// TwinCAT 3 PLC project Untitled1
// ProgramVersion: 3.1.4023.0
// libraries:
//   Tc2_Standard, * (Beckhoff Automation GmbH)
//   Tc2_System, * (Beckhoff Automation GmbH)
//   Tc3_EventLogger, * (Beckhoff Automation GmbH)
//   Tc3_Module, * (Beckhoff Automation GmbH)
//   VisuDialogs, * (System)
//   VisuSymbols,3.5.10.0,System
// project tree:
//   / GlobalTextList.TcGTLO (not stored), PlcTask.TcTTO (not stored), Visualization Manager.TcVMO (not stored)
//   POUs/ MAIN.TcPOU
// real-time tasks:
//   TASK PlcTask: cycle T#10ms, priority 20, ADS port 350
// I/O:
//   DEVICE Device 1 (EtherCAT), AmsNetId 5.112.67.239.2.1
//     Term 7 (EK1200) [EK1200-5000 EtherCAT Power supply (2A E-Bus)]
//       Term 2 (EL4004) [EL4004 4Ch. Ana. Output 0-10V, 12bit]
//       Term 3 (EL4004) [EL4004 4Ch. Ana. Output 0-10V, 12bit]
//       Term 8 (EL3024) [EL3024 4Ch. Ana. Input 4-20mA DIFF]
//       Term 9 (EL3024) [EL3024 4Ch. Ana. Input 4-20mA DIFF]
//       Term 12 (EL1859) [EL1859 8Ch. Dig. Input 24V, 3ms, 8Ch. Dig. Output 24V, 0.5A]
//       Term 13 (EL9011) [EL9011 End Terminal]
// variable links:
//   Untitled1/Untitled1 Instance <-> Device 1 (EtherCAT)/Term 7 (EK1200)/Term 12 (EL1859)
//     PlcTask Inputs/MAIN.EMERGENCY_STOP <-> Channel 1/EMERGENCY STOP
//     PlcTask Inputs/MAIN.Start_Button <-> Channel 2/Start Button
//     PlcTask Inputs/MAIN.Stop_Button <-> Channel 3/Stop Button
//     PlcTask Outputs/MAIN.Motor_Direction <-> Channel 10/Motor Direction
//     PlcTask Outputs/MAIN.Motor_ON_OFF <-> Channel 9/Motor ON/OFF
//   Untitled1/Untitled1 Instance <-> Device 1 (EtherCAT)/Term 7 (EK1200)/Term 2 (EL4004)
//     PlcTask Outputs/MAIN.Flow_Valve_1 <-> AO Outputs Channel 4/Flow_Valve_1
//     PlcTask Outputs/MAIN.Level_Valve_1 <-> AO Outputs Channel 1/Level_Valve_1
//     PlcTask Outputs/MAIN.Level_Valve_2 <-> AO Outputs Channel 2/Level_Valve_2
//     PlcTask Outputs/MAIN.Level_Valve_3 <-> AO Outputs Channel 3/Level_Valve_3
//   Untitled1/Untitled1 Instance <-> Device 1 (EtherCAT)/Term 7 (EK1200)/Term 3 (EL4004)
//     PlcTask Outputs/MAIN.Gas_Valve <-> AO Outputs Channel 1/Gas_Valve
//     PlcTask Outputs/MAIN.Mixer_Valve <-> AO Outputs Channel 2/Mixer_Valve
//     PlcTask Outputs/MAIN.Motor_speed <-> AO Outputs Channel 3/Motor_Speed
//   Untitled1/Untitled1 Instance <-> Device 1 (EtherCAT)/Term 7 (EK1200)/Term 8 (EL3024)
//     PlcTask Inputs/MAIN.Pressure_Differencial_Transmitter_1 <-> AI Standard Channel 1/PDT 1
//     PlcTask Inputs/MAIN.Pressure_Differencial_Transmitter_2 <-> AI Standard Channel 3/PDT 2
//     PlcTask Inputs/MAIN.Pressure_Transmitter_1 <-> AI Standard Channel 2/PT 1
//     PlcTask Inputs/MAIN.Pressure_Transmitter_3 <-> AI Standard Channel 4/PT 3
//   Untitled1/Untitled1 Instance <-> Device 1 (EtherCAT)/Term 7 (EK1200)/Term 9 (EL3024)
//     PlcTask Inputs/MAIN.Level_Transmitter_1 <-> AI Standard Channel 2/ Level Transmitter 1
//     PlcTask Inputs/MAIN.Level_Transmitter_2 <-> AI Standard Channel 3/Level Transmitter 2
//     PlcTask Inputs/MAIN.Pressure_Transmitter_2 <-> AI Standard Channel 1/PT 2
//     PlcTask Inputs/MAIN.Temperature_Transmitter <-> AI Standard Channel 4/Temperature Transmitter

// ---- POUs/MAIN.TcPOU
PROGRAM MAIN
VAR
	//Linking variables to IO cards
	Flow_Valve_1 AT %Q* : INT;
	Level_Valve_1 AT %Q* : INT;
	Level_Valve_2 AT %Q* : INT;
	Level_Valve_3 AT %Q* : INT;
	Gas_Valve AT %Q* : INT;
	Mixer_Valve AT %Q* : INT;
	Motor_speed AT %Q* : INT;
	Motor_ON_OFF AT %Q* :BOOL;
	Motor_Direction AT %Q* :BOOL; 
	Start_Button AT %I* :BOOL;
	Stop_Button AT %I* : BOOL; 
	EMERGENCY_STOP AT %I* : BOOL; 
	Level_Transmitter_1 AT %I* :INT; 
	Level_Transmitter_2 AT %I* :INT; 
	Temperature_Transmitter AT %I* :INT;  
	Pressure_Differencial_Transmitter_1 AT %I* : INT;
	Pressure_Differencial_Transmitter_2 AT %I* : INT;
	Pressure_Transmitter_1 AT %I* : INT ; 
	Pressure_Transmitter_2 AT %I* : INT ; 
	Pressure_Transmitter_3 AT %I* : INT ; 

	
	//User Input as percentage
	Flow_Valve_1_Percentage: INT :=100;
	Level_Valve_1_Percentage: INT    ;
	Level_Valve_2_Percentage: INT;
	Level_Valve_3_Percentage: INT;
	Motor_speed_Percentage: INT; 
	Motor_ON : BOOL ; 
	ON_OFF : STRING(10) := 'OFF' ; 
	
	
	
	
END_VAR



// variable interval for Flow_Valve_1_Percentage  form 0 to 100  
IF Flow_Valve_1_Percentage > 100 THEN
	Flow_Valve_1_Percentage := 100; 
	ELSE IF Flow_Valve_1_Percentage < 0 THEN 
		Flow_Valve_1_Percentage := 0; 
	END_IF
	
END_IF

// variable interval for Level_Valve_1_Percentage  form 0 to 100  
IF Level_Valve_1_Percentage > 100 THEN
	Level_Valve_1_Percentage := 100; 
	ELSE IF Level_Valve_1_Percentage < 0 THEN 
		Level_Valve_1_Percentage := 0; 
	END_IF
	
END_IF

// variable interval for Level_Valve_2_Percentage  form 0 to 100 
IF Level_Valve_2_Percentage > 100 THEN
	Level_Valve_2_Percentage := 100; 
	ELSE IF Level_Valve_2_Percentage < 0 THEN 
		Level_Valve_2_Percentage := 0; 
	END_IF
	
END_IF

// variable interval for Level_Valve_3_Percentage  form 0 to 100 
IF Level_Valve_3_Percentage > 100 THEN
	Level_Valve_3_Percentage := 100; 
	ELSE IF Level_Valve_3_Percentage < 0 THEN 
		Level_Valve_3_Percentage := 0; 
	END_IF
	
END_IF



// variable interval for Motor_speed_Percentage  form 0 to 100 
IF Motor_speed_Percentage > 100 THEN
	Motor_speed_Percentage := 100; 
	ELSE IF Motor_speed_Percentage < 0 THEN 
		Motor_speed_Percentage := 0; 
	END_IF
	
END_IF

// Flow_Valve_1 calibration
Flow_Valve_1 := REAL_TO_INT (262.14*Flow_Valve_1_Percentage +6553 ); 

// Level_Valve_1 calibration
Level_Valve_1 := REAL_TO_INT(262.14*Level_Valve_1_Percentage +6553);

// Level_Valve_2 calibration
Level_Valve_2 := REAL_TO_INT(262.14*Level_Valve_2_Percentage +6553);

// Level_Valve_3 calibration
Level_Valve_3 := REAL_TO_INT(262.14*Level_Valve_3_Percentage +6553);


// Motor_speed calibration
Motor_speed := REAL_TO_INT(262.14*Motor_speed_Percentage +6553);

 
IF Motor_ON_OFF   THEN
    Motor_ON   :=  FALSE;
	ON_OFF  := 'MOTOR: ON' ;
	
ELSE
    Motor_ON  := TRUE;
	ON_OFF  := 'MOTOR: OFF' ;
END_IF

END_PROGRAM
